// TIA Portal V20 export
FUNCTION_BLOCK "Lift_Driver"   // FB5, LAD
{ S7_Optimized_Access := 'TRUE' }
// stored: MemoryReserve 100, SetENOAutomatically false
   VAR_INPUT
      Jog_Forward : Bool;
      Jog_Backward : Bool;
      Velocity : LReal := 50.0;
      Reset : Bool;
      Halt : Bool;
      Power : Bool;
   END_VAR
   VAR
      MC_POWER_Lift { S7_SetPoint := 'True'} : MC_POWER;
      Alarm { S7_SetPoint := 'True'} : Byte;   // X0 - Power, X1 - Reset, X2 - Halt, X3-Jog
   END_VAR
BEGIN

REGION Network 1
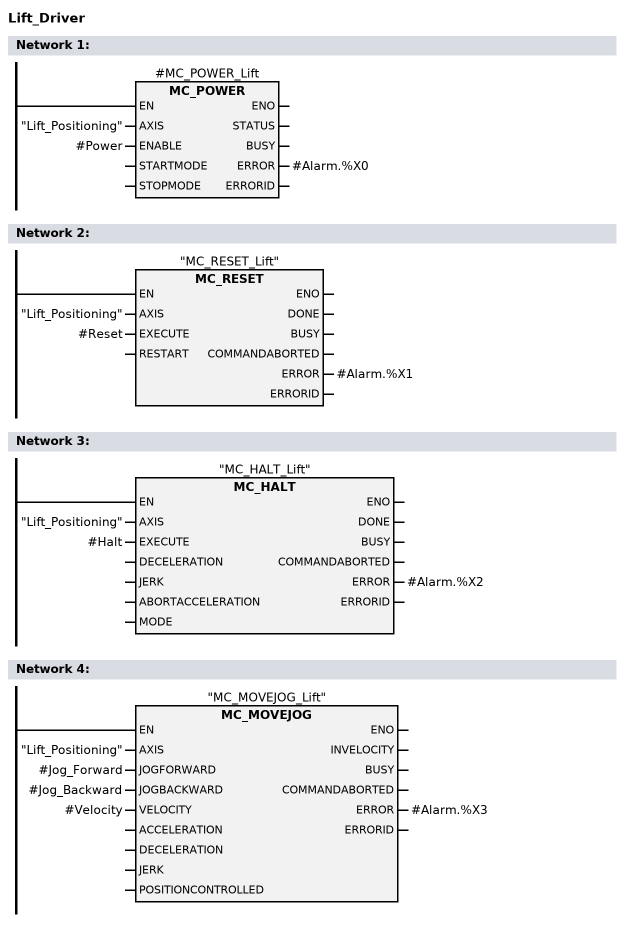
   RUNG wire#powerrail
      #MC_POWER_Lift.MC_POWER(Axis := "Lift_Positioning", Enable := #Power, StartMode :=, StopMode :=, Status =>, Busy =>, Error => #Alarm.%X0, ErrorId =>)
   END_RUNG
   // the same network as SCL:
   #MC_POWER_Lift(Axis := "Lift_Positioning", Enable := #Power, Error => #Alarm.%X0);   // MC_POWER
END_REGION

REGION Network 2
   RUNG wire#powerrail
      "MC_RESET_Lift".MC_RESET(Axis := "Lift_Positioning", Execute := #Reset, Restart :=, Done =>, Busy =>, CommandAborted =>, Error => #Alarm.%X1, ErrorId =>)
   END_RUNG
   // the same network as SCL:
   "MC_RESET_Lift"(Axis := "Lift_Positioning", Execute := #Reset, Error => #Alarm.%X1);   // MC_RESET
END_REGION

REGION Network 3
   RUNG wire#powerrail
      "MC_HALT_Lift".MC_HALT(Axis := "Lift_Positioning", Execute := #Halt, Deceleration :=, Jerk :=, AbortAcceleration :=, Mode :=, Done =>, Busy =>, CommandAborted =>, Error => #Alarm.%X2, ErrorId =>)
   END_RUNG
   // the same network as SCL:
   "MC_HALT_Lift"(Axis := "Lift_Positioning", Execute := #Halt, Error => #Alarm.%X2);   // MC_HALT
END_REGION

REGION Network 4
   RUNG wire#powerrail
      "MC_MOVEJOG_Lift".MC_MOVEJOG(Axis := "Lift_Positioning", JogForward := #Jog_Forward, JogBackward := #Jog_Backward, Velocity := #Velocity, Acceleration :=, Deceleration :=, Jerk :=, PositionControlled :=, InVelocity =>, Busy =>, CommandAborted =>, Error => #Alarm.%X3, ErrorId =>)
   END_RUNG
   // the same network as SCL:
   "MC_MOVEJOG_Lift"(Axis := "Lift_Positioning",   // MC_MOVEJOG
                     JogForward := #Jog_Forward,
                     JogBackward := #Jog_Backward,
                     Velocity := #Velocity,
                     Error => #Alarm.%X3);
END_REGION
END_FUNCTION_BLOCK
